{attribute addProperty BoxType "EL2014-0000-0016"}
{attribute addProperty Id "DIG_Diag_InputsAT %I*DIG_Diag_Inputs_B107C8FA1620DIG_Inputs_DeviceAT %I*DIG_Inputs_Device_07359F0E3240DIG_OutputsAT %Q*DIG_Outputs_276DFED340.50WcStateAT %I*WcState_98A4DF7520.250InfoDataAT %I*InfoData_BC63D37F80100"}
{attribute addProperty CRC "2162136907"}
{attribute addProperty SizeInBites "134"}
{attribute addProperty SizeInBytes "16.75"}
TYPE EL2014_B1F56BCC :
STRUCT
	{attribute addProperty Name "DIG_Diag_Inputs"}
	DIG_Diag_Inputs : DIG_Diag_Inputs_B107C8FA;
	{attribute addProperty Name "DIG_Inputs_Device"}
	DIG_Inputs_Device : DIG_Inputs_Device_07359F0E;
	{attribute addProperty Name "DIG_Outputs"}
	DIG_Outputs : DIG_Outputs_276DFED3;
	{attribute addProperty Name "WcState"}
	WcState : WcState_98A4DF75;
	{attribute addProperty Name "InfoData"}
	InfoData : InfoData_BC63D37F;
END_STRUCT
END_TYPE

(* stored: Version 1.2.0.0, ProductVersion 3.1.4024.9
   DUT EL2014_B1F56BCC: Id {367cee80-6f85-4893-942f-2b7c99f51527} *)
